{attribute 'GeneratedUsingTerminal: EL2252--0000'}
{attribute addProperty BoxType "EL2252--0000"}
{attribute addProperty Id "StartTimeAT %Q*UDINT4"}
{attribute addProperty CRC "2630553169"}
{attribute addProperty Size "4"}
TYPE DC_Sync_Start_9CCB0E51 EXTENDS OutputBase_10CEE7DE :
STRUCT
	{attribute addProperty Name "StartTime"}
	StartTime AT %Q* : UDINT;
END_STRUCT
END_TYPE

(* stored: Version 1.2.0.0, ProductVersion 3.1.4024.9
   DUT DC_Sync_Start_9CCB0E51: Id {df377a65-ebf7-49f0-9241-212b8e5b592c} *)
